{attribute 'qualified_only'}
VAR_GLOBAL
	{attribute 'OPC.UA.DA' := '1'}
	{attribute 'OPC.UA.DA.Access' := '1'}
	{attribute 'init_namespace'} 
	Name : STRING(255);	
END_VAR

(* stored: Version 1.1.0.1
   GVL CurrentNamespace_1: Id {004d2be3-b47a-4802-a4dd-c17d706125fb} *)
